# EPICS substitutions: apps/jscalerApp/Db/jscalers_TDCFTOF1_TRIG.substitutions
file "db/jscaler_channel.db" {
pattern { CrNo,CrName,Sl,Ch,Det,Sys,Element,CScode,Thresh,Mode,Counts }
{ "05","TDCFTOF1","20","15","TRIG","CAEN","SEC1","5125","15","271","15" }
}
